# B&R Automation Studio project heating_io
Automation Studio 3.0.80.42
